{attribute 'pack_mode' := '1'}
    {attribute 'OPC.UA.DA' := '1'}
    {attribute 'OPC.UA.DA.StructuredType' := '1'}
    (*
    ST_RW_PlcInfo_HMI_IgnitionExp
    ==================================================
    Generated from Ignition UDT: RW_PLC_Info
    Total tags: 15
    Generated on: 2025-09-15 12:47:18
    *)
    TYPE ST_RW_PlcInfo_HMI_IgnitionExp :
    STRUCT
        {attribute 'OPC.UA.DA' := '1'}
        {attribute 'OPC.UA.DA.Access' := '1'}
        KW_Device_SecondsInError : SINT := 0;		// Read-only tag
        {attribute 'OPC.UA.DA' := '1'}
        {attribute 'OPC.UA.DA.Access' := '1'}
        FirmwareVersion : STRING := '';		// Read-only tag
        {attribute 'OPC.UA.DA' := '1'}
        {attribute 'OPC.UA.DA.Access' := '1'}
        CurrentCycleTime : REAL := 0.0;		// Read-only tag
        {attribute 'OPC.UA.DA' := '1'}
        {attribute 'OPC.UA.DA.Access' := '1'}
        CycleTimeLimit : REAL := 0.0;		// Read-only tag
        {attribute 'OPC.UA.DA' := '1'}
        KW_ForceSymbolReload : BOOL := FALSE;

        {attribute 'OPC.UA.DA' := '1'}
        {attribute 'OPC.UA.DA.Access' := '1'}
        KW_Device_ScanRateMs : DINT := 0;		// Read-only tag
        {attribute 'OPC.UA.DA' := '1'}
        {attribute 'OPC.UA.DA.Access' := '1'}
        KW_Device_Error : BOOL := FALSE;		// Read-only tag
        {attribute 'OPC.UA.DA' := '1'}
        {attribute 'OPC.UA.DA.Access' := '1'}
        KW_Device_Enabled : BOOL := FALSE;		// Read-only tag
        {attribute 'OPC.UA.DA' := '1'}
        {attribute 'OPC.UA.DA.Access' := '1'}
        KW_Device_ScanMode : STRING := '';		// Read-only tag
        {attribute 'OPC.UA.DA' := '1'}
        {attribute 'OPC.UA.DA.Access' := '1'}
        MinimumCycleTime : REAL := 0.0;		// Read-only tag

        {attribute 'OPC.UA.DA' := '1'}
        {attribute 'OPC.UA.DA.Access' := '1'}
        IPAddress : STRING := '';		// Read-only tag
        {attribute 'OPC.UA.DA' := '1'}
        {attribute 'OPC.UA.DA.Access' := '1'}
        KW_Device_Description : STRING := '';		// Read-only tag
        {attribute 'OPC.UA.DA' := '1'}
        {attribute 'OPC.UA.DA.Access' := '1'}
        Model : STRING := '';		// Read-only tag
        {attribute 'OPC.UA.DA' := '1'}
        {attribute 'OPC.UA.DA.Access' := '1'}
        OB1Runtime : REAL := 0.0;		// Read-only tag
        {attribute 'OPC.UA.DA' := '1'}
        {attribute 'OPC.UA.DA.Access' := '1'}
        KW_Device_ActiveTagCount : DINT := 0;		// Read-only tag
    END_STRUCT
    END_TYPE

(* stored: Version 1.1.0.1
   DUT ST_RW_PlcInfo_HMI_IgnitionExp: Id {30cb1036-8fb9-4165-b735-175b510f00f5} *)
